Omron Sysmac Studio project Test3 (Sysmac Studio 1.56.0.64011, StandardProject)

# Controller new_Controller_0: NX1P2-1040DT1 version 1.16
Task PrimaryTask (priority 4, period or condition 2000): Program0

VAR_GLOBAL
    BIO_Input_Bit_00 : BOOL;  (* at BuiltInIO://cpu/#0/Input_Bit_00 *)
    BIO_Input_Bit_01 : BOOL;  (* at BuiltInIO://cpu/#0/Input_Bit_01 *)
    BIO_Input_Bit_02 : BOOL;  (* at BuiltInIO://cpu/#0/Input_Bit_02 *)
    Start : BOOL;
    Stop : BOOL;
    Çıkış : BOOL;
    Motor : BOOL;
    Start2 : BOOL;
    Motorİleri : BOOL;
    Motor_İleri : BOOL;
    Motor_Geri : BOOL;
END_VAR

PROGRAM Program0
VAR_EXTERNAL
    Start : BOOL;
    Stop : BOOL;
    Çıkış : BOOL;
    Motor : BOOL;
    BIO_Input_Bit_00 : BOOL;
    BIO_Input_Bit_01 : BOOL;
    BIO_Input_Bit_02 : BOOL;
    Start2 : BOOL;
    Motorİleri : BOOL;
    Motor_İleri : BOOL;
    Motor_Geri : BOOL;
END_VAR

(* Section InOut: ladder, written here as Structured Text *)

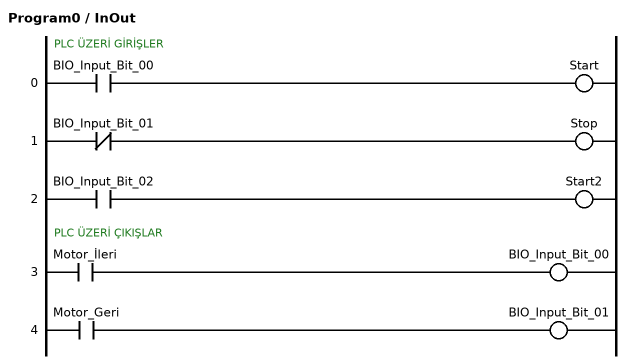
(* Rung 0: PLC ÜZERİ GİRİŞLER *)
Start := BIO_Input_Bit_00;
(* Rung 1 *)
Stop := NOT BIO_Input_Bit_01;
(* Rung 2 *)
Start2 := BIO_Input_Bit_02;
(* Rung 3: PLC ÜZERİ ÇIKIŞLAR *)
BIO_Input_Bit_00 := Motor_İleri;
(* Rung 4 *)
BIO_Input_Bit_01 := Motor_Geri;

(* Section Section1: ladder, written here as Structured Text *)

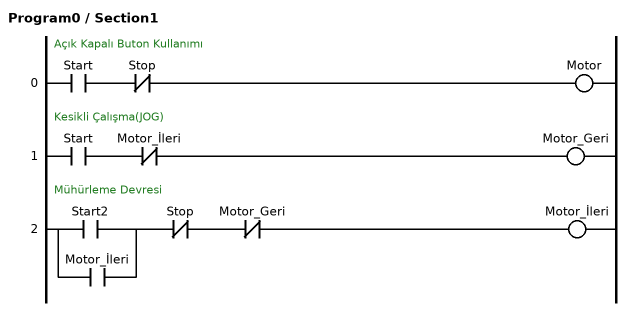
(* Rung 0: Açık Kapalı Buton Kullanımı *)
Motor := Start AND NOT Stop;
(* Rung 1: Kesikli Çalışma(JOG) *)
Motor_Geri := Start AND NOT Motor_İleri;
(* Rung 2: Mühürleme Devresi *)
Motor_İleri := (Start2 OR Motor_İleri) AND NOT Stop AND NOT Motor_Geri;
END_PROGRAM